FUNCTION_BLOCK FB_Dynamic_Stack IMPLEMENTS I_Stack
VAR_INPUT
END_VAR
VAR_OUTPUT
END_VAR
VAR
END_VAR

{warning 'add method implementation '}
METHOD Peek : T_DATA_TYPE
END_METHOD

{warning 'add method implementation '}
METHOD Pop
END_METHOD

{warning 'add method implementation '}
METHOD Push
VAR_INPUT
	Data	: T_DATA_TYPE;
END_VAR
END_METHOD

{warning 'add method implementation '}
METHOD Show
END_METHOD

END_FUNCTION_BLOCK

(* stored: Version 1.1.0.1, ProductVersion 3.1.4024.4
   POU FB_Dynamic_Stack: Id {6794da22-5d0c-48e6-b3a8-88d57cbb32b9}, SpecialFunc None
   Method Peek: Id {2eb5ed08-a9b0-4fdc-a4fc-6c6b26d9bcd6}
   Method Pop: Id {bbedc7b5-0295-4ee8-ac30-b3b8281ee07b}
   Method Push: Id {1192dd04-d4fd-4b27-af4d-9615dea0bc87}
   Method Show: Id {4fb0df02-3ae9-4af9-9983-b8822a8b4e2e} *)
